// TIA Portal V20 export
DATA_BLOCK "DB_ScannerComm"   // DB126
// stored: InstanceOfName FB_ScannerComm, InstanceOfType FB
"FB_ScannerComm"
   // VAR_INPUT
   //    iInit : Bool;
   //    iReady : Bool;
   //    iStatus : DInt;
   //    iStatusDescription : String;
   //    iCheckNumber : Byte;
   //    iPartOnFixture : Bool;
   //    iStationNumber : Byte;
   //    iHoleNumber : DInt;
   //    iJobListName : String;
   //    iJobName : DInt;
   //    iMeasureZ : LReal;
   // END_VAR
   // VAR_OUTPUT
   //    oIsFirstJobOfPiece : Bool;
   //    oStationNumber : Byte;
   //    oHoleNumber : DInt;
   //    oJobListName : String;
   //    oJobName : String;
   //    oMeasureZ : LReal;
   //    oBadPart : Bool;
   //    oGoodPart : Bool;
   //    oEndOfJob : Bool;
   // END_VAR
   // VAR_IN_OUT
   //    ioRequestJob_NC : Bool;
   //    ioReady_NC : Bool;
   //    ioCheckNumber : Byte;
   //    ioRequestJob : Bool;
   // END_VAR
   // VAR
   //    sRT_PartOnFixture : R_TRIG;
   //    sRT_Ready { S7_SetPoint := 'True'} : R_TRIG;
   //    sEndOfJob { S7_SetPoint := 'True'} : Bool;
   //    sRT_RequestJob_NC : R_TRIG;
   //    sJobListName { S7_SetPoint := 'True'} : String;
   //    sJobName : String;
   //    sJobInProgress : Bool;
   // END_VAR
BEGIN
END_DATA_BLOCK
